// TIA Portal V17 export
// export: Created 2025-03-07T09:16:38.4737309Z, ExportSetting WithDefaults, DisplayName Totally Integrated Automation Portal, DisplayVersion V17 Update 8, DisplayName TIA Portal Openness, DisplayVersion V17 Update 8, DisplayName TIA Portal Version Control Interface, DisplayVersion V17, DisplayName SINAMICS Startdrive Advanced, DisplayVersion V17 SP2, DisplayName SINAMICS Startdrive G110M, G120, G120C, G120D, G120P, G115D, DisplayVersion V17 SP2, DisplayName SINAMICS Startdrive G130, G150, S120, S150, SINAMICS MV, S210, DisplayVersion V17 SP2, DisplayName STEP 7 Professional, DisplayVersion V17 Update 8, DisplayName SINUMERIK ONE STEP 7 Toolbox, DisplayVersion V17 Update 12, DisplayName SINUMERIK 840D sl STEP 7 Toolbox, DisplayVersion V17 Update 12, DisplayName STEP 7 Safety, DisplayVersion V17 Update 6, DisplayName WinCC Advanced, DisplayVersion V17 Update 8
DATA_BLOCK "DB2400_DBB_VALUES"   // DB2400
{ S7_Optimized_Access := 'FALSE'; DB_Accessible_From_OPC_UA := 'FALSE' }
AUTHOR : ETXETAR
VERSION : 1.0
// stored: AutoNumber false, DBAccessibleFromOPCUA false, DBAccessibleFromWebserver true, IsOnlyStoredInLoadMemory false, IsWriteProtectedInAS false
   VAR RETAIN
      DBB_DBW_DBD_VAL_0 : UInt := 0;   // MACHINE CNC CYCLE UNIT 01 STATION 0 ($A_DBB[0])
      DBB_DBW_DBD_VAL_1 : UInt := 1;
      DBB_DBW_DBD_VAL_2 : UInt := 2;   // MACHINE CNC CYCLE UNIT 01 STATION 3 ($A_DBB[2])
      DBB_DBW_DBD_VAL_3 : UInt := 3;
      DBB_DBW_DBD_VAL_4 : UInt := 4;   // MACHINE CNC CYCLE UNIT 01 STATION 4 ($A_DBB[4])
      DBB_DBW_DBD_VAL_5 : UInt := 5;
      DBB_DBW_DBD_VAL_6 : UInt := 6;   // MACHINE CNC CYCLE UNIT 02 STATION 0 ($A_DBB[6])
      DBB_DBW_DBD_VAL_7 : UInt := 7;
      DBB_DBW_DBD_VAL_8 : UInt := 8;   // MACHINE CNC CYCLE UNIT 02 STATION 2 ($A_DBB[8])
      DBB_DBW_DBD_VAL_9 : UInt := 9;
      DBB_DBW_DBD_VAL_10 : UInt := 10;   // MACHINE CNC CYCLE UNIT 02 STATION 3 ($A_DBB[9])
      DBB_DBW_DBD_VAL_11 : UInt := 11;
      DBB_DBW_DBD_VAL_12 : UInt := 12;   // MACHINE CNC CYCLE UNIT 02 STATION 4 ($A_DBB[9])
      DBB_DBW_DBD_VAL_14 : UInt := 14;   // MACHINE CNC CYCLE UNIT 03 STATION 0 ($A_DBB[14])
      DBB_DBW_DBD_VAL_19 : UInt := 19;
      DBB_DBW_DBD_VAL_20 : UInt := 20;   // FIXTURE NUMBER IN UNIT 01 STATION 1 ($A_DBB[20])
      DBB_DBW_DBD_VAL_22 : UInt := 22;   // FIXTURE NUMBER IN UNIT 02 STATION 1 ($A_DBB[22])
      DBB_DBW_DBD_VAL_23 : UInt := 23;
      DBB_DBW_DBD_VAL_24 : UInt := 24;
      DBB_DBW_DBD_VAL_30 : UInt := 30;   // PART TYPE ($A_DBB[30])
      DBB_DBW_DBD_VAL_31 : UInt := 31;
      DBB_DBW_DBD_VAL_34 : UInt := 34;
      DBB_DBW_DBD_VAL_35 : UInt := 35;
      DBB_DBW_DBD_VAL_40 : UInt := 40;   // FIXTURE 1 MACHINING MEMORY TO FULL DEPTH UNIT 01R ($A_DBB[40])
      DBB_DBW_DBD_VAL_41 : UInt := 41;   // FIXTURE 1 MACHINING MEMORY TO FULL DEPTH UNIT 01L ($A_DBB[41])
      DBB_DBW_DBD_VAL_44 : UInt := 44;   // FIXTURE 1 BACK CHAMFERS TRACER ($A_DBB[44])
      DBB_DBW_DBD_VAL_45 : UInt := 45;   // FIXTURE 1 TAPPING TRACER ($A_DBB[45])
      DBB_DBW_DBD_VAL_48 : UInt := 48;   // FIXTURE 2 MACHINING MEMORY TO FULL DEPTH UNIT 01R ($A_DBB[48])
      DBB_DBW_DBD_VAL_49 : UInt := 49;   // FIXTURE 2 MACHINING MEMORY TO FULL DEPTH UNIT 01L ($A_DBB[49])
      DBB_DBW_DBD_VAL_52 : UInt := 52;   // FIXTURE 2 BACK CHAMFERS TRACER ($A_DBB[52])
      DBB_DBW_DBD_VAL_53 : UInt := 53;   // FIXTURE 2 TAPPING TRACER ($A_DBB[53])
      DBB_DBW_DBD_VAL_56 : UInt := 56;   // FIXTURE 1 CLAMP STATUS ($A_DBB[56])
      DBB_DBW_DBD_VAL_57 : UInt := 57;   // FIXTURE 2 CLAMP STATUS ($A_DBB[57])
      DBB_DBW_DBD_VAL_58 : UInt := 58;   // PART SEATED CLAMP RECOVERY UNIT 01R ($A_DBB[58])
      DBB_DBW_DBD_VAL_59 : UInt := 59;   // PART SEATED CLAMP RECOVERY UNIT 01L ($A_DBB[59])
      DBB_DBW_DBD_VAL_60 : UInt := 60;   // AXIS W SAFETY MOVE ($A_DBB[60])
      DBB_DBW_DBD_VAL_61 : UInt := 61;   // AXIS B POSITIONS ($A_DBB[61])
      DBB_DBW_DBD_VAL_62 : UInt := 62;   // AXIS B IN POSITION TO LOAD ($A_DBB[62])
      DBB_DBW_DBD_VAL_64 : UInt := 64;   // MEASURE PROBE ALARM CODE ($A_DBB[64])
      DBB_DBW_DBD_VAL_65 : UInt := 65;   // MEASUREMENT FRECUENCY ($A_DBB[65])
      DBB_DBW_DBD_VAL_66 : UInt := 66;   // RESET GUD CYCLE VARIABLES ($A_DBB[66])
      DBB_DBW_DBD_VAL_67 : UInt := 67;   // CYCLE SELECTION CEMB ENABLE ($A_DBB[67])
      DBB_DBW_DBD_VAL_70 : UInt := 70;   // MQL VARIANT UNIT 01R ($A_DBB[70])
      DBB_DBW_DBD_VAL_71 : UInt := 71;   // MQL VARIANT UNIT 01L ($A_DBB[71])
      DBB_DBW_DBD_VAL_75 : UInt := 75;   // RFID ZONE TO WRITE IN TOOL HOLDER CHIP UNIT 01R ($A_DBB[75])
      DBB_DBW_DBD_VAL_76 : UInt := 76;   // RFID ZONE TO WRITE IN TOOL HOLDER CHIP UNIT 01L ($A_DBB[76])
      DBB_DBW_DBD_VAL_77 : UInt := 77;   // RFID ZONE TO WRITE IN TOOL HOLDER CHIP ($A_DBB[77])
      DBB_DBW_DBD_VAL_80 : UInt := 80;   // TAG ERROR UNIT 01R ($A_DBB[80])
      DBB_DBW_DBD_VAL_81 : UInt := 81;   // TAG ERROR UNIT 01L ($A_DBB[81])
      DBB_DBW_DBD_VAL_100 : UInt := 100;   // TOOL CLAMPING DIFFERENCE SP11 ($A_DBB[100])
      DBB_DBW_DBD_VAL_101 : UInt := 101;   // TOOL CLAMPING DIFFERENCE SP12 ($A_DBB[101])
      DBB_DBW_DBD_VAL_102 : UInt := 102;   // TOOL CLAMPING DIFFERENCE SP13 ($A_DBB[102])
      DBB_DBW_DBD_VAL_103 : UInt := 103;   // TOOL CLAMPING DIFFERENCE SP14 ($A_DBB[103])
      DBB_DBW_DBD_VAL_110 : UInt := 110;   // TOOL CLAMPING DIFFERENCE SP21 ($A_DBB[110])
      DBB_DBW_DBD_VAL_111 : UInt := 111;   // TOOL CLAMPING DIFFERENCE SP22 ($A_DBB[111])
      DBB_DBW_DBD_VAL_112 : UInt := 112;   // TOOL CLAMPING DIFFERENCE SP23 ($A_DBB[112])
      DBB_DBW_DBD_VAL_113 : UInt := 113;   // TOOL CLAMPING DIFFERENCE SP24 ($A_DBB[113])
      DBB_DBW_DBD_VAL_120 : UInt := 120;   // MAGAZINE MEMORY ALARM UNIT 01R ($A_DBB[120])
      DBB_DBW_DBD_VAL_121 : UInt := 121;   // MAGAZINE MEMORY ALARM TYPE UNIT 01R ($A_DBB[121])
      DBB_DBW_DBD_VAL_122 : UInt := 122;   // MAGAZINE TOOL FAULTED UNIT 01R ($A_DBB[122])
      DBB_DBW_DBD_VAL_123 : UInt := 123;   // MAGAZINE TOOL IN ERROR DATA UNIT 01R ($A_DBB[123])
      DBB_DBW_DBD_VAL_125 : UInt := 125;   // MAGAZINE MEMORY ALARM UNIT 01L ($A_DBB[125])
      DBB_DBW_DBD_VAL_126 : UInt := 126;   // MAGAZINE MEMORY ALARM TYPE UNIT 01L ($A_DBB[126])
      DBB_DBW_DBD_VAL_127 : UInt := 127;   // MAGAZINE TOOL FAULTED UNIT 01L ($A_DBB[127])
      DBB_DBW_DBD_VAL_128 : UInt := 128;   // MAGAZINE TOOL IN ERROR DATA UNIT 01L ($A_DBB[128])
      DBB_DBW_DBD_VAL_150 : UInt := 150;   // BK MIKRO MAGAZINE POSITION SP11 ($A_DBB[150])
      DBB_DBW_DBD_VAL_151 : UInt := 151;   // BK MIKRO MAGAZINE POSITION SP12 ($A_DBB[151])
      DBB_DBW_DBD_VAL_152 : UInt := 152;   // BK MIKRO MAGAZINE POSITION SP13 ($A_DBB[152])
      DBB_DBW_DBD_VAL_153 : UInt := 153;   // BK MIKRO MAGAZINE POSITION SP14 ($A_DBB[153])
      DBB_DBW_DBD_VAL_154 : UInt := 154;   // BK MIKRO MAGAZINE POSITION SP21 ($A_DBB[154])
      DBB_DBW_DBD_VAL_155 : UInt := 155;   // BK MIKRO MAGAZINE POSITION SP22 ($A_DBB[155])
      DBB_DBW_DBD_VAL_156 : UInt := 156;   // BK MIKRO MAGAZINE POSITION SP23 ($A_DBB[156])
      DBB_DBW_DBD_VAL_157 : UInt := 157;   // BK MIKRO MAGAZINE POSITION SP24 ($A_DBB[157])
      DBB_DBW_DBD_VAL_160 : UInt := 160;   // UNIT 01 POWDER FEEDER 1 CARRIER GAS NOMINAL LINE 1
      DBB_DBW_DBD_VAL_164 : UInt := 164;   // UNIT 01 POWDER FEEDER 1 CARRIER GAS NOMINAL LINE 2
      DBB_DBW_DBD_VAL_168 : UInt := 168;   // UNIT 01 POWDER FEEDER 1 DISK SPEED NOMINAL LINE 1
      DBB_DBW_DBD_VAL_172 : UInt := 172;   // UNIT 01 POWDER FEEDER 1 DISK SPEED NOMINAL LINE 2
      DBB_DBW_DBD_VAL_176 : UInt := 176;   // UNIT 01 POWDER FEEDER 1 STIRRER SPEED NOMINAL LINE 1
      DBB_DBW_DBD_VAL_180 : UInt := 180;   // UNIT 01 POWDER FEEDER 1 STIRRER SPEED NOMINAL LINE 2
      DBB_DBW_DBD_VAL_184 : UInt := 184;   // UNIT 01 POWDER FEEDER 1 HOPPER TEMPERATURE NOMINAL LINE 1
      DBB_DBW_DBD_VAL_188 : UInt := 188;   // UNIT 01 POWDER FEEDER 1 HOPPER TEMPERATURE NOMINAL LINE 2
      DBB_DBW_DBD_VAL_200 : UInt := 200;   // UNIT 02 POWDER FEEDER 1 CARRIER GAS NOMINAL LINE 1
      DBB_DBW_DBD_VAL_204 : UInt := 204;   // UNIT 02 POWDER FEEDER 1 CARRIER GAS NOMINAL LINE 2
      DBB_DBW_DBD_VAL_208 : UInt := 208;   // UNIT 02 POWDER FEEDER 1 DISK SPEED NOMINAL LINE 1
      DBB_DBW_DBD_VAL_212 : UInt := 212;   // UNIT 02 POWDER FEEDER 1 DISK SPEED NOMINAL LINE 2
      DBB_DBW_DBD_VAL_216 : UInt := 216;   // UNIT 02 POWDER FEEDER 1 STIRRER SPEED NOMINAL LINE 1
      DBB_DBW_DBD_VAL_220 : UInt := 220;   // UNIT 02 POWDER FEEDER 1 STIRRER SPEED NOMINAL LINE 2
      DBB_DBW_DBD_VAL_224 : UInt := 224;   // UNIT 02 POWDER FEEDER 1 HOPPER TEMPERATURE NOMINAL LINE 1
      DBB_DBW_DBD_VAL_228 : UInt := 228;   // UNIT 02 POWDER FEEDER 1 HOPPER TEMPERATURE NOMINAL LINE 2
      DBB_DBW_DBD_VAL_240 : UInt := 240;   // UNIT 02 POWDER FEEDER 2 CARRIER GAS NOMINAL LINE 1
      DBB_DBW_DBD_VAL_244 : UInt := 244;   // UNIT 02 POWDER FEEDER 2 CARRIER GAS NOMINAL LINE 2
      DBB_DBW_DBD_VAL_248 : UInt := 248;   // UNIT 02 POWDER FEEDER 2 DISK SPEED NOMINAL LINE 1
      DBB_DBW_DBD_VAL_252 : UInt := 252;   // UNIT 02 POWDER FEEDER 2 DISK SPEED NOMINAL LINE 2
      DBB_DBW_DBD_VAL_256 : UInt := 256;   // UNIT 02 POWDER FEEDER 2 STIRRER SPEED NOMINAL LINE 1
      DBB_DBW_DBD_VAL_260 : UInt := 260;   // UNIT 02 POWDER FEEDER 2 STIRRER SPEED NOMINAL LINE 2
      DBB_DBW_DBD_VAL_264 : UInt := 264;   // UNIT 02 POWDER FEEDER 2 HOPPER TEMPERATURE NOMINAL LINE 1
      DBB_DBW_DBD_VAL_268 : UInt := 268;   // UNIT 02 POWDER FEEDER 2 HOPPER TEMPERATURE NOMINAL LINE 2
      DBB_DBW_DBD_VAL_504 : UInt := 504;   // UNIT 01LASER POWER ($A_DBB[504])
      DBB_DBW_DBD_VAL_506 : UInt := 506;   // UNIT 01 LASER PROCESSING (0=CORE / 1=RING / 3=BRIGHTLINE WELD) ($A_DBB[506])
      DBB_DBW_DBD_VAL_508 : UInt := 508;   // UNIT 01 LASER POWER PORTION CORE (%) ($A_DBB[508])
      DBB_DBW_DBD_VAL_514 : UInt := 514;   // UNIT 02 LASER POWER ($A_DBB[514])
      DBB_DBW_DBD_VAL_516 : UInt := 516;   // UNIT 02 LASER PROCESSING (0=CORE / 1=RING / 3=BRIGHTLINE WELD) ($A_DBB[516])
      DBB_DBW_DBD_VAL_518 : UInt := 518;   // UNIT 02 LASER POWER PORTION CORE (%) ($A_DBB[518])
      DBB_DBW_DBD_VAL_1000 : UInt := 1000;   // UNIT 01 FIXTURE 1 PART A QUALITY STATUS ($A_DBB[1000])
      DBB_DBW_DBD_VAL_1001 : UInt := 1001;   // UNIT 01 FIXTURE 1 PART A PROCESS STATUS ($A_DBB[1001])
      DBB_DBW_DBD_VAL_1002 : UInt := 1002;   // UNIT 01 FIXTURE 1 PART C ($A_DBB[1002])
      DBB_DBW_DBD_VAL_1003 : UInt := 1003;   // UNIT 01 FIXTURE 1 PART D ($A_DBB[1003])
      DBB_DBW_DBD_VAL_1006 : UInt := 1006;   // UNIT 01 FIXTURE 2 PART A QUALITY STATUS ($A_DBB[1006])
      DBB_DBW_DBD_VAL_1007 : UInt := 1007;   // UNIT 01 FIXTURE 2 PART A PROCESS STATUS ($A_DBB[1007])
      DBB_DBW_DBD_VAL_1008 : UInt := 1008;   // UNIT 01 FIXTURE 2 PART C ($A_DBB[1008])
      DBB_DBW_DBD_VAL_1009 : UInt := 1009;   // UNIT 01 FIXTURE 2 PART D ($A_DBB[1009])
      DBB_DBW_DBD_VAL_1012 : UInt := 1012;   // UNIT 01 FIXTURE 3 PART A QUALITY STATUS ($A_DBB[1012])
      DBB_DBW_DBD_VAL_1013 : UInt := 1013;   // UNIT 01 FIXTURE 3 PART A PROCESS STATUS ($A_DBB[1013])
      DBB_DBW_DBD_VAL_1014 : UInt := 1014;   // UNIT 01 FIXTURE 3 PART C ($A_DBB[1014])
      DBB_DBW_DBD_VAL_1015 : UInt := 1015;   // UNIT 01 FIXTURE 3 PART D ($A_DBB[1015])
      DBB_DBW_DBD_VAL_1018 : UInt := 1018;   // UNIT 01 FIXTURE 4 PART A QUALITY STATUS ($A_DBB[1018])
      DBB_DBW_DBD_VAL_1019 : UInt := 1019;   // UNIT 01 FIXTURE 4 PART A PROCESS STATUS ($A_DBB[1019])
      DBB_DBW_DBD_VAL_1020 : UInt := 1020;   // UNIT 01 FIXTURE 4 PART C ($A_DBB[1020])
      DBB_DBW_DBD_VAL_1021 : UInt := 1021;   // UNIT 01 FIXTURE 4 PART D ($A_DBB[1021])
      DBB_DBW_DBD_VAL_1024 : UInt := 1024;   // UNIT 02 FIXTURE 1 PART A QUALITY STATUS ($A_DBB[1024])
      DBB_DBW_DBD_VAL_1025 : UInt := 1025;   // UNIT 02 FIXTURE 1 PART A PROCESS STATUS ($A_DBB[1025])
      DBB_DBW_DBD_VAL_1026 : UInt := 1026;   // UNIT 02 FIXTURE 1 PART C ($A_DBB[1026])
      DBB_DBW_DBD_VAL_1027 : UInt := 1027;   // UNIT 02 FIXTURE 1 PART D ($A_DBB[1027])
      DBB_DBW_DBD_VAL_1030 : UInt := 1030;   // UNIT 02 FIXTURE 2 PART A QUALITY STATUS ($A_DBB[1030])
      DBB_DBW_DBD_VAL_1031 : UInt := 1031;   // UNIT 02 FIXTURE 2 PART A PROCESS STATUS ($A_DBB[1031])
      DBB_DBW_DBD_VAL_1032 : UInt := 1032;   // UNIT 02 FIXTURE 2 PART C ($A_DBB[1032])
      DBB_DBW_DBD_VAL_1033 : UInt := 1033;   // UNIT 02 FIXTURE 2 PART D ($A_DBB[1033])
      DBB_DBW_DBD_VAL_1036 : UInt := 1036;   // UNIT 02 FIXTURE 3 PART A QUALITY STATUS ($A_DBB[1036])
      DBB_DBW_DBD_VAL_1037 : UInt := 1037;   // UNIT 02 FIXTURE 3 PART A PROCESS STATUS ($A_DBB[1037])
      DBB_DBW_DBD_VAL_1038 : UInt := 1038;   // UNIT 02 FIXTURE 3 PART C ($A_DBB[1038])
      DBB_DBW_DBD_VAL_1039 : UInt := 1039;   // UNIT 02 FIXTURE 3 PART D ($A_DBB[1039])
      DBB_DBW_DBD_VAL_1042 : UInt := 1042;   // UNIT 02 FIXTURE 4 PART A QUALITY STATUS ($A_DBB[1042])
      DBB_DBW_DBD_VAL_1043 : UInt := 1043;   // UNIT 02 FIXTURE 4 PART A PROCESS STATUS ($A_DBB[1043])
      DBB_DBW_DBD_VAL_1044 : UInt := 1044;   // UNIT 02 FIXTURE 4 PART C ($A_DBB[1044])
      DBB_DBW_DBD_VAL_1045 : UInt := 1045;   // UNIT 02 FIXTURE 4 PART D ($A_DBB[1045])
      DBB_DBW_DBD_VAL_1048 : UInt := 1048;   // UNIT 01 STATION 1 PART A QUALITY STATUS ($A_DBB[1048])
      DBB_DBW_DBD_VAL_1049 : UInt := 1049;   // UNIT 01 STATION 1 PART A PROCESS STATUS ($A_DBB[1049])
      DBB_DBW_DBD_VAL_1050 : UInt := 1050;   // UNIT 01 STATION 1 PART C ($A_DBB[1050])
      DBB_DBW_DBD_VAL_1051 : UInt := 1051;   // UNIT 01 STATION 1 PART D ($A_DBB[1051])
      DBB_DBW_DBD_VAL_1200 : UInt := 1200;   // CLEAN TOOL HOLDERS UNIT 01R ($A_DBB[1200])
      DBB_DBW_DBD_VAL_1201 : UInt := 1201;   // CLEAN TOOL HOLDERS SEQUENCE DONE UNIT 01R ($A_DBB[1201])
      DBB_DBW_DBD_VAL_1204 : UInt := 1204;   // CLEAN TOOL HOLDERS UNIT 01L ($A_DBB[1204])
      DBB_DBW_DBD_VAL_1205 : UInt := 1205;   // CLEAN TOOL HOLDERS SEQUENCE DONE UNIT 01L ($A_DBB[1205])
      DBB_DBW_DBD_VAL_1250 : UInt := 1250;   // WAIT CHANNEL 1 ($A_DBB[1250])
      DBB_DBW_DBD_VAL_1272 : UInt := 1272;   // UNIT 01 AXIS X13 ACTUAL SPEED ($A_DBB[1272])
      DBB_DBW_DBD_VAL_1276 : UInt := 1276;   // FIXTURE 1 PART A FLANGE Y ($A_DBB[1276])
      DBB_DBW_DBD_VAL_1280 : UInt := 1280;   // FIXTURE 1 PART A POST X ($A_DBB[1280])
      DBB_DBW_DBD_VAL_1284 : UInt := 1284;   // FIXTURE 1 PART A POST Y ($A_DBB[1284])
      DBB_DBW_DBD_VAL_1288 : UInt := 1288;   // FIXTURE 1 PART B FLANGE X ($A_DBB[1288])
      DBB_DBW_DBD_VAL_1292 : UInt := 1292;   // UNIT 01 SPINDLE C13 ACTUAL SPEED ($A_DBB[1292])
      DBB_DBW_DBD_VAL_1296 : UInt := 1296;   // FIXTURE 1 PART B POST X ($A_DBB[1296])
      DBB_DBW_DBD_VAL_1300 : UInt := 1300;   // FIXTURE 1 PART B POST Y ($A_DBB[1300])
      DBB_DBW_DBD_VAL_1352 : UInt := 1352;   // UNIT 02 AXIS X23 ACTUAL SPEED ($A_DBB[1352])
      DBB_DBW_DBD_VAL_1356 : UInt := 1356;   // FIXTURE 2 PART A FLANGE Y ($A_DBB[1356])
      DBB_DBW_DBD_VAL_1360 : UInt := 1360;   // FIXTURE 2 PART A POST X ($A_DBB[1360])
      DBB_DBW_DBD_VAL_1364 : UInt := 1364;   // FIXTURE 2 PART A POST Y ($A_DBB[1364])
      DBB_DBW_DBD_VAL_1368 : UInt := 1368;   // FIXTURE 2 PART B FLANGE X ($A_DBB[1368])
      DBB_DBW_DBD_VAL_1372 : UInt := 1372;   // UNIT 02 SPINDLE C23 ACTUAL SPEED ($A_DBB[1372])
      DBB_DBW_DBD_VAL_1376 : UInt := 1376;   // FIXTURE 2 PART B POST X ($A_DBB[1376])
      DBB_DBW_DBD_VAL_1380 : UInt := 1380;   // FIXTURE 2 PART B POST Y ($A_DBB[1380])
      DBB_DBW_DBD_VAL_1450 : UInt := 1450;   // NC TEST PROGRAM AXIS SELECTION ($A_DBB[1450])
      DBB_DBW_DBD_VAL_1452 : UInt := 1452;   // SERVICE POSITION PROGRAM SELECTION ($A_DBB[1452])
      DBB_DBW_DBD_VAL_1454 : UInt := 1454;   // SPEED FOR SP11. VIBRATION ANALYSIS ($A_DBB54
      DBB_DBW_DBD_VAL_1456 : UInt := 1456;   // SPEED FOR SP12. VIBRATION ANALYSIS ($A_DBB[1456])
      DBB_DBW_DBD_VAL_1458 : UInt := 1458;   // TIME FOR ANALYSIS. VIBRATION ANALYSIS UNIT 01R ($A_DBB[1458])
      DBB_DBW_DBD_VAL_1460 : UInt := 1460;   // TIME FOR START. VIBRATION ANALYSIS UNIT 01R ($A_DBB[1460])
      DBB_DBW_DBD_VAL_1462 : UInt := 1462;   // SPEED FOR SP21. VIBRATION ANALYSIS ($A_DBB[1462])
      DBB_DBW_DBD_VAL_1464 : UInt := 1464;   // SPEED FOR SP22. VIBRATION ANALYSIS ($A_DBB[1464])
      DBB_DBW_DBD_VAL_1466 : UInt := 1466;   // TIME FOR ANALYSIS. VIBRATION ANALYSIS UNIT 01L ($A_DBB[1466])
      DBB_DBW_DBD_VAL_1468 : UInt := 1468;   // TIME FOR START. VIBRATION ANALYSIS UNIT 01L ($A_DBB[1468])
      DBB_DBW_DBD_VAL_1500 : UInt := 1500;   // TOOL NAME. TOOL MAGAZINE 01R ($A_DBB[1500])
      DBB_DBW_DBD_VAL_1532 : UInt := 1532;   // DUPLO NUMBER. TOOL MAGAZINE 01R ($A_DBB[1532])
      DBB_DBW_DBD_VAL_1534 : UInt := 1534;   // LOCATION TYPE. TOOL MAGAZINE 01R ($A_DBB[1534])
      DBB_DBW_DBD_VAL_1536 : UInt := 1536;   // SIEMENS TOOL STATUS. TOOL MAGAZINE 01R ($A_DBB[1536])
      DBB_DBW_DBD_VAL_1538 : UInt := 1538;   // TYPE OF TOOL MONITORING. TOOL MAGAZINE 01R ($A_DBB[1538])
      DBB_DBW_DBD_VAL_1540 : UInt := 1540;   // CHECK TOOL BROKEN. TOOL MAGAZINE 01R ($A_DBB[1540])
      DBB_DBW_DBD_VAL_1542 : UInt := 1542;   // NUMBER OF CUTTING EDGES. TOOL MAGAZINE 01R ($A_DBB[1542])
      DBB_DBW_DBD_VAL_1544 : UInt := 1544;   // OEM 1. TOOL MAGAZINE 01R ($A_DBB[1544])
      DBB_DBW_DBD_VAL_1548 : UInt := 1548;   // OEM 2. TOOL MAGAZINE 01R ($A_DBB[1548])
      DBB_DBW_DBD_VAL_1552 : UInt := 1552;   // OEM 3. TOOL MAGAZINE 01R ($A_DBB[1552])
      DBB_DBW_DBD_VAL_1556 : UInt := 1556;   // OEM 4. TOOL MAGAZINE 01R ($A_DBB[1556])
      DBB_DBW_DBD_VAL_1560 : UInt := 1560;   // OEM 5. TOOL MAGAZINE 01R ($A_DBB[1560])
      DBB_DBW_DBD_VAL_1564 : UInt := 1564;   // OEM 6. TOOL MAGAZINE 01R ($A_DBB[1564])
      DBB_DBW_DBD_VAL_1568 : UInt := 1568;   // OEM 7. TOOL MAGAZINE 01R ($A_DBB[1568])
      DBB_DBW_DBD_VAL_1572 : UInt := 1572;   // OEM 8. TOOL MAGAZINE 01R ($A_DBB[1572])
      DBB_DBW_DBD_VAL_1576 : UInt := 1576;   // OEM 9. TOOL MAGAZINE 01R ($A_DBB[1576])
      DBB_DBW_DBD_VAL_1580 : UInt := 1580;   // OEM 10. TOOL MAGAZINE 01R ($A_DBB[1580])
      DBB_DBW_DBD_VAL_1584 : UInt := 1584;   // TOOL TYPE EDGE 1. TOOL MAGAZINE 01R ($A_DBB[1584])
      DBB_DBW_DBD_VAL_1586 : UInt := 1586;   // CUTTING POSITION EDGE 1. TOOL MAGAZINE 01R ($A_DBB[1586])
      DBB_DBW_DBD_VAL_1588 : UInt := 1588;   // TOOL LENGTH 1 EDGE 1. TOOL MAGAZINE 01R ($A_DBB[1588])
      DBB_DBW_DBD_VAL_1592 : UInt := 1592;   // TOOL LENGTH 2 EDGE 1. TOOL MAGAZINE 01R ($A_DBB[1592])
      DBB_DBW_DBD_VAL_1596 : UInt := 1596;   // TOOL LENGTH 3 EDGE 1. TOOL MAGAZINE 01R ($A_DBB[1596])
      DBB_DBW_DBD_VAL_1600 : UInt := 1600;   // TOOL RADIUS EDGE 1. TOOL MAGAZINE 01R ($A_DBB[1600])
      DBB_DBW_DBD_VAL_1604 : UInt := 1604;   // TOOL PITCH EDGE 1. TOOL MAGAZINE 01R ($A_DBB[1604])
      DBB_DBW_DBD_VAL_1608 : UInt := 1608;   // WEAR LENGTH EDGE 1. TOOL MAGAZINE 01R ($A_DBB[1608])
      DBB_DBW_DBD_VAL_1620 : UInt := 1620;   // WEAR RADIUS EDGE 1. TOOL MAGAZINE 01R ($A_DBB[1620])
      DBB_DBW_DBD_VAL_1645 : UInt := 1644;
      DBB_DBW_DBD_VAL_1644 : UInt := 1644;   // WARNING TOOL LIFE EDGE 1. TOOL MAGAZINE 01R ($A_DBB[1644])
      DBB_DBW_DBD_VAL_1648 : UInt := 1648;   // ACTUAL TOOL LIFE EDGE 1. TOOL MAGAZINE 01R ($A_DBB[1648])
      DBB_DBW_DBD_VAL_1652 : UInt := 1652;   // SET POINT QUANTITY EDGE 1. TOOL MAGAZINE 01R ($A_DBB[1652])
      DBB_DBW_DBD_VAL_1664 : UInt := 1664;   // TOOL TYPE EDGE 2. TOOL MAGAZINE 01R ($A_DBB[1664])
      DBB_DBW_DBD_VAL_1666 : UInt := 1666;   // CUTTING POSITION EDGE 2. TOOL MAGAZINE 01R ($A_DBB[1666])
      DBB_DBW_DBD_VAL_1668 : UInt := 1668;   // TOOL LENGTH 1 EDGE 2. TOOL MAGAZINE 01R ($A_DBB[1668])
      DBB_DBW_DBD_VAL_1672 : UInt := 1672;   // TOOL LENGTH 2 EDGE 2. TOOL MAGAZINE 01R ($A_DBB[1672])
      DBB_DBW_DBD_VAL_1676 : UInt := 1676;   // TOOL LENGTH 3 EDGE 2. TOOL MAGAZINE 01R ($A_DBB[1676])
      DBB_DBW_DBD_VAL_1680 : UInt := 1680;   // TOOL RADIUS EDGE 2. TOOL MAGAZINE 01R ($A_DBB[1680])
      DBB_DBW_DBD_VAL_1684 : UInt := 1684;   // TOOL PITCH EDGE 2. TOOL MAGAZINE 01R ($A_DBB[1684])
      DBB_DBW_DBD_VAL_1688 : UInt := 1688;   // WEAR LENGTH EDGE 2. TOOL MAGAZINE 01R ($A_DBB[1688])
      DBB_DBW_DBD_VAL_1700 : UInt := 1700;   // UNIT_01_NOOZLE_SURFACE_DISTANCE
      DBB_DBW_DBD_VAL_1704 : UInt := 1704;   // UNIT_02_NOOZLE_SURFACE_DISTANCE
      DBB_DBW_DBD_VAL_1724 : UInt := 1724;   // WARNING TOOL LIFE EDGE 2. TOOL MAGAZINE 01R ($A_DBB[1724])
      DBB_DBW_DBD_VAL_1728 : UInt := 1728;   // ACTUAL TOOL LIFE EDGE 2. TOOL MAGAZINE 01R ($A_DBB[1728])
      DBB_DBW_DBD_VAL_1732 : UInt := 1732;   // SET POINT QUANTITY EDGE 2. TOOL MAGAZINE 01R ($A_DBB[1732])
      DBB_DBW_DBD_VAL_1744 : UInt := 1744;   // TOOL TYPE EDGE 3. TOOL MAGAZINE 01R ($A_DBB[1744])
      DBB_DBW_DBD_VAL_1746 : UInt := 1746;   // CUTTING POSITION EDGE 3. TOOL MAGAZINE 01R ($A_DBB[1746])
      DBB_DBW_DBD_VAL_1748 : UInt := 1748;   // TOOL LENGTH 1 EDGE 3. TOOL MAGAZINE 01R ($A_DBB[1748])
      DBB_DBW_DBD_VAL_1752 : UInt := 1752;   // TOOL LENGTH 2 EDGE 3. TOOL MAGAZINE 01R ($A_DBB[1752])
      DBB_DBW_DBD_VAL_1756 : UInt := 1756;   // TOOL LENGTH 3 EDGE 3. TOOL MAGAZINE 01R ($A_DBB[1756])
      DBB_DBW_DBD_VAL_1760 : UInt := 1760;   // TOOL RADIUS EDGE 3. TOOL MAGAZINE 01R ($A_DBB[1760])
      DBB_DBW_DBD_VAL_1764 : UInt := 1764;   // TOOL PITCH EDGE 3. TOOL MAGAZINE 01R ($A_DBB[1764])
      DBB_DBW_DBD_VAL_1768 : UInt := 1768;   // WEAR LENGTH EDGE 3. TOOL MAGAZINE 01R ($A_DBB[1768])
      DBB_DBW_DBD_VAL_1780 : UInt := 1780;   // WEAR RADIUS EDGE 3. TOOL MAGAZINE 01R ($A_DBB[1780])
      DBB_DBW_DBD_VAL_1804 : UInt := 1804;   // WARNING TOOL LIFE EDGE 3. TOOL MAGAZINE 01R ($A_DBB[1804])
      DBB_DBW_DBD_VAL_1808 : UInt := 1808;   // ACTUAL TOOL LIFE EDGE 3. TOOL MAGAZINE 01R ($A_DBB[1808])
      DBB_DBW_DBD_VAL_1812 : UInt := 1812;   // SET POINT QUANTITY EDGE 3. TOOL MAGAZINE 01R ($A_DBB[1812])
      DBB_DBW_DBD_VAL_1824 : UInt := 1824;   // TOOL TYPE EDGE 4. TOOL MAGAZINE 01R ($A_DBB[1824])
      DBB_DBW_DBD_VAL_1826 : UInt := 1826;   // CUTTING POSITION EDGE 4. TOOL MAGAZINE 01R ($A_DBB[1826])
      DBB_DBW_DBD_VAL_1828 : UInt := 1828;   // TOOL LENGTH 1 EDGE 4. TOOL MAGAZINE 01R ($A_DBB[1828])
      DBB_DBW_DBD_VAL_1832 : UInt := 1832;   // TOOL LENGTH 2 EDGE 4. TOOL MAGAZINE 01R ($A_DBB[1832])
      DBB_DBW_DBD_VAL_1836 : UInt := 1836;   // TOOL LENGTH 3 EDGE 4. TOOL MAGAZINE ($A_DBB[1836])
      DBB_DBW_DBD_VAL_1840 : UInt := 1840;   // TOOL RADIUS EDGE 4. TOOL MAGAZINE 01R ($A_DBB[1840])
      DBB_DBW_DBD_VAL_1844 : UInt := 1844;   // TOOL PITCH EDGE 4. TOOL MAGAZINE 01R ($A_DBB[1844])
      DBB_DBW_DBD_VAL_1848 : UInt := 1848;   // WEAR LENGTH EDGE 4. TOOL MAGAZINE 01R ($A_DBB[1848])
      DBB_DBW_DBD_VAL_1860 : UInt := 1860;   // WEAR RADIUS EDGE 4. TOOL MAGAZINE 01R ($A_DBB[1860])
      DBB_DBW_DBD_VAL_1884 : UInt := 1884;   // WARNING TOOL LIFE EDGE 4. TOOL MAGAZINE 01R ($A_DBB[1884])
      DBB_DBW_DBD_VAL_1888 : UInt := 1888;   // ACTUAL TOOL LIFE EDGE 4. TOOL MAGAZINE 01R ($A_DBB[1888])
      DBB_DBW_DBD_VAL_1892 : UInt := 1892;   // SET POINT QUANTITY EDGE 4. TOOL MAGAZINE 01R ($A_DBB[1892])
      DBB_DBW_DBD_VAL_1904 : UInt := 1904;   // TOOL TYPE EDGE 5. TOOL MAGAZINE 01R ($A_DBB[1904])
      DBB_DBW_DBD_VAL_1906 : UInt := 1906;   // CUTTING POSITION EDGE 5. TOOL MAGAZINE 01R ($A_DBB[1906])
      DBB_DBW_DBD_VAL_1908 : UInt := 1908;   // TOOL LENGTH 1 EDGE 5. TOOL MAGAZINE 01R ($A_DBB[1908])
      DBB_DBW_DBD_VAL_1912 : UInt := 1912;   // TOOL LENGTH 2 EDGE 5. TOOL MAGAZINE 01R ($A_DBB[1912])
      DBB_DBW_DBD_VAL_1916 : UInt := 1916;   // TOOL LENGTH 3 EDGE 5. TOOL MAGAZINE 01R ($A_DBB[1916])
      DBB_DBW_DBD_VAL_1920 : UInt := 1920;   // TOOL RADIUS EDGE 5. TOOL MAGAZINE 01R ($A_DBB[1920])
      DBB_DBW_DBD_VAL_1924 : UInt := 1924;   // TOOL PITCH EDGE 5. TOOL MAGAZINE 01R ($A_DBB[1924])
      DBB_DBW_DBD_VAL_1928 : UInt := 1928;   // WEAR LENGTH EDGE 5. TOOL MAGAZINE 01R ($A_DBB[1928])
      DBB_DBW_DBD_VAL_1940 : UInt := 1940;   // WEAR RADIUS EDGE 5. TOOL MAGAZINE 01R ($A_DBB[1940])
      DBB_DBW_DBD_VAL_1964 : UInt := 1964;   // WARNING TOOL LIFE EDGE 5. TOOL MAGAZINE 01R ($A_DBB[1964])
      DBB_DBW_DBD_VAL_1968 : UInt := 1968;   // ACTUAL TOOL LIFE EDGE 5. TOOL MAGAZINE 01R ($A_DBB[1968])
      DBB_DBW_DBD_VAL_1972 : UInt := 1972;   // SET POINT QUANTITY EDGE 5. TOOL MAGAZINE 01R ($A_DBB[1972])
      DBB_DBW_DBD_VAL_1984 : UInt := 1984;   // GM SPINDLE NUMBER 01R ($A_DBB[1984])
      DBB_DBW_DBD_VAL_2000 : UInt := 2000;   // TOOL NAME. TOOL MAGAZINE 01L ($A_DBB[2000])
      DBB_DBW_DBD_VAL_2032 : UInt := 2032;   // DUPLO NUMBER. TOOL MAGAZINE 01L ($A_DBB[2032])
      DBB_DBW_DBD_VAL_2034 : UInt := 2034;   // LOCATION TYPE. TOOL MAGAZINE 01L ($A_DBB[2034])
      DBB_DBW_DBD_VAL_2036 : UInt := 2036;   // SIEMENS TOOL STATUS. TOOL MAGAZINE 01L ($A_DBB[2036])
      DBB_DBW_DBD_VAL_2038 : UInt := 2038;   // TYPE OF TOOL MONITORING. TOOL MAGAZINE 01L ($A_DBB[2038])
      DBB_DBW_DBD_VAL_2040 : UInt := 2040;   // CHECK TOOL BROKEN. TOOL MAGAZINE 01L ($A_DBB[2040])
      DBB_DBW_DBD_VAL_2042 : UInt := 2042;   // NUMBER OF CUTTING EDGES. TOOL MAGAZINE 01L ($A_DBB[2042])
      DBB_DBW_DBD_VAL_2044 : UInt := 2044;   // OEM 1. TOOL MAGAZINE 01L ($A_DBB[2044])
      DBB_DBW_DBD_VAL_2048 : UInt := 2048;   // OEM 2. TOOL MAGAZINE 01L ($A_DBB[2048])
      DBB_DBW_DBD_VAL_2052 : UInt := 2052;   // OEM 3. TOOL MAGAZINE 01L ($A_DBB[2052])
      DBB_DBW_DBD_VAL_2056 : UInt := 2056;   // OEM 4. TOOL MAGAZINE 01L ($A_DBB[2056])
      DBB_DBW_DBD_VAL_2060 : UInt := 2060;   // OEM 5. TOOL MAGAZINE 01L ($A_DBB[2060])
      DBB_DBW_DBD_VAL_2064 : UInt := 2064;   // OEM 6. TOOL MAGAZINE 01L ($A_DBB[2064])
      DBB_DBW_DBD_VAL_2068 : UInt := 2068;   // OEM 7. TOOL MAGAZINE 01L ($A_DBB[2068])
      DBB_DBW_DBD_VAL_2072 : UInt := 2072;   // OEM 8. TOOL MAGAZINE 01L ($A_DBB[2072])
      DBB_DBW_DBD_VAL_2076 : UInt := 2076;   // OEM 9. TOOL MAGAZINE 01L ($A_DBB[2076])
      DBB_DBW_DBD_VAL_2080 : UInt := 2080;   // OEM 10. TOOL MAGAZINE 01L ($A_DBB[2080])
      DBB_DBW_DBD_VAL_2084 : UInt := 2084;   // TOOL TYPE EDGE 1. TOOL MAGAZINE 01L ($A_DBB[2084])
      DBB_DBW_DBD_VAL_2086 : UInt := 2086;   // CUTTING POSITION EDGE 1. TOOL MAGAZINE 01L ($A_DBB[2086])
      DBB_DBW_DBD_VAL_2088 : UInt := 2088;   // TOOL LENGTH 1 EDGE 1. TOOL MAGAZINE 01L ($A_DBB[2088])
      DBB_DBW_DBD_VAL_2092 : UInt := 2092;   // TOOL LENGTH 2 EDGE 1. TOOL MAGAZINE 01L ($A_DBB[2092])
      DBB_DBW_DBD_VAL_2096 : UInt := 2096;   // TOOL LENGTH 3 EDGE 1. TOOL MAGAZINE 01L ($A_DBB[209])
      DBB_DBW_DBD_VAL_2100 : UInt := 2100;   // TOOL RADIUS EDGE 1. TOOL MAGAZINE 01L ($A_DBB[2100])
      DBB_DBW_DBD_VAL_2104 : UInt := 2104;   // TOOL PITCH EDGE 1. TOOL MAGAZINE 01L ($A_DBB[2104])
      DBB_DBW_DBD_VAL_2108 : UInt := 2108;   // WEAR LENGTH EDGE 1. TOOL MAGAZINE 01L ($A_DBB[2108])
      DBB_DBW_DBD_VAL_2120 : UInt := 2120;   // WEAR RADIUS EDGE 1. TOOL MAGAZINE 01L ($A_DBB[2120])
      DBB_DBW_DBD_VAL_2144 : UInt := 2144;   // WARNING TOOL LIFE EDGE 1. TOOL MAGAZINE 01L ($A_DBB[2144])
      DBB_DBW_DBD_VAL_2148 : UInt := 2148;   // ACTUAL TOOL LIFE EDGE 1. TOOL MAGAZINE 01L ($A_DBB[2148])
      DBB_DBW_DBD_VAL_2152 : UInt := 2152;   // SET POINT QUANTITY EDGE 1. TOOL MAGAZINE 01L ($A_DBB[2152])
      DBB_DBW_DBD_VAL_2164 : UInt := 2164;   // TOOL TYPE EDGE 2. TOOL MAGAZINE 01L ($A_DBB[2164])
      DBB_DBW_DBD_VAL_2166 : UInt := 2166;   // CUTTING POSITION EDGE 2. TOOL MAGAZINE 01L ($A_DBB[2166])
      DBB_DBW_DBD_VAL_2168 : UInt := 2168;   // TOOL LENGTH 1 EDGE 2. TOOL MAGAZINE 01L ($A_DBB[2168])
      DBB_DBW_DBD_VAL_2172 : UInt := 2172;   // TOOL LENGTH 2 EDGE 2. TOOL MAGAZINE 01L ($A_DBB[2172])
      DBB_DBW_DBD_VAL_2176 : UInt := 2176;   // TOOL LENGTH 3 EDGE 2. TOOL MAGAZINE 01L ($A_DBB[2176])
      DBB_DBW_DBD_VAL_2180 : UInt := 2180;   // TOOL RADIUS EDGE 2. TOOL MAGAZINE 01L ($A_DBB[2180])
      DBB_DBW_DBD_VAL_2184 : UInt := 2184;   // TOOL PITCH EDGE 2. TOOL MAGAZINE 01L ($A_DBB[2184])
      DBB_DBW_DBD_VAL_2188 : UInt := 2188;   // WEAR LENGTH EDGE 2. TOOL MAGAZINE 01L ($A_DBB[2188])
      DBB_DBW_DBD_VAL_2200 : UInt := 2200;   // WEAR RADIUS EDGE 2. TOOL MAGAZINE 01L ($A_DBB[2200])
      DBB_DBW_DBD_VAL_2224 : UInt := 2224;   // WARNING TOOL LIFE EDGE 2. TOOL MAGAZINE 01L ($A_DBB[2224])
      DBB_DBW_DBD_VAL_2228 : UInt := 2228;   // ACTUAL TOOL LIFE EDGE 2. TOOL MAGAZINE 01L ($A_DBB[2228])
      DBB_DBW_DBD_VAL_2232 : UInt := 2232;   // SET POINT QUANTITY EDGE 2. TOOL MAGAZINE 01L ($A_DBB[2232])
      DBB_DBW_DBD_VAL_2244 : UInt := 2244;   // TOOL TYPE EDGE 3. TOOL MAGAZINE 01L ($A_DBB[2244])
      DBB_DBW_DBD_VAL_2246 : UInt := 2246;   // CUTTING POSITION EDGE 3. TOOL MAGAZINE 01L ($A_DBB[2246])
      DBB_DBW_DBD_VAL_2248 : UInt := 2248;   // TOOL LENGTH 1 EDGE 3. TOOL MAGAZINE 01L ($A_DBB[2248])
      DBB_DBW_DBD_VAL_2252 : UInt := 2252;   // TOOL LENGTH 2 EDGE 3. TOOL MAGAZINE 01L ($A_DBB[2252])
      DBB_DBW_DBD_VAL_2256 : UInt := 2256;   // TOOL LENGTH 3 EDGE 3. TOOL MAGAZINE 01L ($A_DBB[2256])
      DBB_DBW_DBD_VAL_2260 : UInt := 2260;   // TOOL RADIUS EDGE 3. TOOL MAGAZINE 01L ($A_DBB[2260])
      DBB_DBW_DBD_VAL_2264 : UInt := 2264;   // TOOL PITCH EDGE 3. TOOL MAGAZINE 01L ($A_DBB[2264])
      DBB_DBW_DBD_VAL_2268 : UInt := 2268;   // WEAR LENGTH EDGE 3. TOOL MAGAZINE 01L ($A_DBB[2268])
      DBB_DBW_DBD_VAL_2280 : UInt := 2280;   // WEAR RADIUS EDGE 3. TOOL MAGAZINE 01L ($A_DBB[2280])
      DBB_DBW_DBD_VAL_2304 : UInt := 2304;   // WARNING TOOL LIFE EDGE 3. TOOL MAGAZINE 01L ($A_DBB[2304])
      DBB_DBW_DBD_VAL_2308 : UInt := 2308;   // ACTUAL TOOL LIFE EDGE 3. TOOL MAGAZINE 01L ($A_DBB[2308])
      DBB_DBW_DBD_VAL_2312 : UInt := 2312;   // SET POINT QUANTITY EDGE 3. TOOL MAGAZINE 01L ($A_DBB[2312])
      DBB_DBW_DBD_VAL_2324 : UInt := 2324;   // TOOL TYPE EDGE 4. TOOL MAGAZINE 01L ($A_DBB[2324])
      DBB_DBW_DBD_VAL_2326 : UInt := 2326;   // CUTTING POSITION EDGE 4. TOOL MAGAZINE 01L ($A_DBB[2326])
      DBB_DBW_DBD_VAL_2328 : UInt := 2328;   // TOOL LENGTH 1 EDGE 4. TOOL MAGAZINE 01L ($A_DBB[2328])
      DBB_DBW_DBD_VAL_2332 : UInt := 2332;   // TOOL LENGTH 2 EDGE 4. TOOL MAGAZINE 01L ($A_DBB[2332])
      DBB_DBW_DBD_VAL_2336 : UInt := 2336;   // TOOL LENGTH 3 EDGE 4. TOOL MAGAZINE 01L ($A_DBB[2336])
      DBB_DBW_DBD_VAL_2340 : UInt := 2340;   // TOOL RADIUS EDGE 4. TOOL MAGAZINE 01L ($A_DBB[2340])
      DBB_DBW_DBD_VAL_2344 : UInt := 2344;   // TOOL PITCH EDGE 4. TOOL MAGAZINE 01L ($A_DBB[2344])
      DBB_DBW_DBD_VAL_2348 : UInt := 2348;   // WEAR LENGTH EDGE 4. TOOL MAGAZINE 01L ($A_DBB[2348])
      DBB_DBW_DBD_VAL_2360 : UInt := 2360;   // WEAR RADIUS EDGE 4. TOOL MAGAZINE 01L ($A_DBB[2360])
      DBB_DBW_DBD_VAL_2384 : UInt := 2384;   // WARNING TOOL LIFE EDGE 4. TOOL MAGAZINE 01L ($A_DBB[2384])
      DBB_DBW_DBD_VAL_2388 : UInt := 2388;   // ACTUAL TOOL LIFE EDGE 4. TOOL MAGAZINE 01L ($A_DBB[2388])
      DBB_DBW_DBD_VAL_2392 : UInt := 2392;   // SET POINT QUANTITY EDGE 4. TOOL MAGAZINE 01L ($A_DBB[2392])
      DBB_DBW_DBD_VAL_2404 : UInt := 2404;   // TOOL TYPE EDGE 5. TOOL MAGAZINE 01L ($A_DBB[2404])
      DBB_DBW_DBD_VAL_2406 : UInt := 2406;   // CUTTING POSITION EDGE 5. TOOL MAGAZINE 01L ($A_DBB[2406])
      DBB_DBW_DBD_VAL_2408 : UInt := 2408;   // TOOL LENGTH 1 EDGE 5. TOOL MAGAZINE 01L ($A_DBB[2408])
      DBB_DBW_DBD_VAL_2412 : UInt := 2412;   // TOOL LENGTH 2 EDGE 5. TOOL MAGAZINE 01L ($A_DBB[2412])
      DBB_DBW_DBD_VAL_2416 : UInt := 2416;   // TOOL LENGTH 3 EDGE 5. TOOL MAGAZINE 01L ($A_DBB[2416])
      DBB_DBW_DBD_VAL_2420 : UInt := 2420;   // TOOL RADIUS EDGE 5. TOOL MAGAZINE 01L ($A_DBB[2420])
      DBB_DBW_DBD_VAL_2424 : UInt := 2424;   // TOOL PITCH EDGE 5. TOOL MAGAZINE 01L ($A_DBB[2424)
      DBB_DBW_DBD_VAL_2428 : UInt := 2428;   // WEAR LENGTH EDGE 5. TOOL MAGAZINE 01L ($A_DBB[2428])
      DBB_DBW_DBD_VAL_2440 : UInt := 2440;   // WEAR RADIUS EDGE 5. TOOL MAGAZINE 01L ($A_DBB[2440])
      DBB_DBW_DBD_VAL_2464 : UInt := 2464;   // WARNING TOOL LIFE EDGE 5. TOOL MAGAZINE 01L ($A_DBB[2464])
      DBB_DBW_DBD_VAL_2468 : UInt := 2468;   // ACTUAL TOOL LIFE EDGE 5. TOOL MAGAZINE 01L ($A_DBB[2468])
      DBB_DBW_DBD_VAL_2472 : UInt := 2472;   // SET POINT QUANTITY EDGE 5. TOOL MAGAZINE 01L ($A_DBB[2472])
      DBB_DBW_DBD_VAL_2484 : UInt := 2484;   // GM SPINDLE NUMBER 01L ($A_DBB[2484])
      DBB_DBW_DBD_VAL_3000 : UInt := 3000;   // CRASH BORE MEASURE POINT 1 ($A_DBB[3000])
      DBB_DBW_DBD_VAL_3004 : UInt := 3004;   // CRASH BORE MEASURE POINT 2 ($A_DBB[3004])
      DBB_DBW_DBD_VAL_3008 : UInt := 3008;   // CRASH BORE MEASURE POINT 3 ($A_DBB[3008])
      DBB_DBW_DBD_VAL_3012 : UInt := 3012;   // CRASH BORE MEASURE POINT 4 ($A_DBB3012)]
      DBB_DBW_DBD_VAL_3016 : UInt := 3016;   // CRASH BORE MEASURE POINT 5 ($A_DBB[3016])
      DBB_DBW_DBD_VAL_3020 : UInt := 3020;   // CRASH BORE MEASURE POINT 6 ($A_DBB[3020])
      DBB_DBW_DBD_VAL_3024 : UInt := 3024;   // CRASH BORE MEASURE POINT 7X ($A_DBB[3024])
      DBB_DBW_DBD_VAL_3028 : UInt := 3028;   // CRASH BORE MEASURE POINT 7Y ($A_DBB[3028])
      DBB_DBW_DBD_VAL_3032 : UInt := 3032;   // CRASH BORE MEASURE POINT 8X ($A_DBB[3032])
      DBB_DBW_DBD_VAL_3036 : UInt := 3036;   // CRASH BORE MEASURE POINT 8Y ($A_DBB[3036])
      DBB_DBW_DBD_VAL_3200 : UInt := 3200;   // MEASURING PROBE PART A 1 ($A_DBB[3200])
      DBB_DBW_DBD_VAL_3204 : UInt := 3204;   // MEASURING PROBE PART A 2 ($A_DBB[3204])
      DBB_DBW_DBD_VAL_3208 : UInt := 3208;   // MEASURING PROBE PART B 1 ($A_DBB[3208])
      DBB_DBW_DBD_VAL_3212 : UInt := 3212;   // MEASURING PROBE PART B 2 ($A_DBB[3212])
      DBB_DBW_DBD_VAL_3216 : UInt := 3216;   // MEASURING PROBE PART C 1 ($A_DBB[3216])
      DBB_DBW_DBD_VAL_3220 : UInt := 3220;   // MEASURING PROBE PART C 2 ($A_DBB[3220])
      DBB_DBW_DBD_VAL_3224 : UInt := 3224;   // MEASURING PROBE PART A1 1 ($A_DBB[3224])
      DBB_DBW_DBD_VAL_3228 : UInt := 3228;   // MEASURING PROBE PART A1 2 ($A_DBB[3228])
      DBB_DBW_DBD_VAL_3232 : UInt := 3232;   // MEASURING PROBE PART B1 1 ($A_DBB[3232])
      DBB_DBW_DBD_VAL_3236 : UInt := 3236;   // MEASURING PROBE PART B1 2 ($A_DBB[3236])
      DBB_DBW_DBD_VAL_3240 : UInt := 3240;   // MEASURING PROBE PART C1 1 ($A_DBB[3240])
      DBB_DBW_DBD_VAL_3244 : UInt := 3244;   // MEASURING PROBE PART C1 2 ($A_DBB[3244])
      DBB_DBW_DBD_VAL_3248 : UInt := 3248;   // MEASURING PROBE PART A2 1 ($A_DBB[3248])
      DBB_DBW_DBD_VAL_3252 : UInt := 3252;   // MEASURING PROBE PART A2 2 ($A_DBB[3252])
      DBB_DBW_DBD_VAL_3256 : UInt := 3256;   // MEASURING PROBE PART B2 1 ($A_DBB[3256])
      DBB_DBW_DBD_VAL_3260 : UInt := 3260;   // MEASURING PROBE PART B2 2 ($A_DBB[3260])
      DBB_DBW_DBD_VAL_3264 : UInt := 3264;   // MEASURING PROBE PART C2 1 ($A_DBB[3264])
      DBB_DBW_DBD_VAL_3268 : UInt := 3268;   // MEASURING PROBE PART C2 2 ($A_DBB[3268])
      DBB_DBW_DBD_VAL_3400 : UInt := 3400;   // TORQUE AXIS SP11 ($A_DBB[3400])
      DBB_DBW_DBD_VAL_3404 : UInt := 3404;   // TORQUE AXIS SP12 ($A_DBB[3404])
      DBB_DBW_DBD_VAL_3408 : UInt := 3408;   // TORQUE AXIS SP13 ($A_DBB[3408])
      DBB_DBW_DBD_VAL_3412 : UInt := 3412;   // TORQUE AXIS SP14 ($A_DBB[3412])
      DBB_DBW_DBD_VAL_3416 : UInt := 3416;   // TORQUE AXIS SP15 ($A_DBB[3416])
      DBB_DBW_DBD_VAL_3420 : UInt := 3420;   // TORQUE AXIS SP16 ($A_DBB[3420])
      DBB_DBW_DBD_VAL_3424 : UInt := 3424;   // TORQUE AXIS SP21 ($A_DBB[3424])
      DBB_DBW_DBD_VAL_3428 : UInt := 3428;   // TORQUE AXIS SP22 ($A_DBB[3428])
      DBB_DBW_DBD_VAL_3432 : UInt := 3432;   // TORQUE AXIS SP23 ($A_DBB[3432])
      DBB_DBW_DBD_VAL_3436 : UInt := 3436;   // TORQUE AXIS SP24 ($A_DBB[3436])
      DBB_DBW_DBD_VAL_3440 : UInt := 3440;   // TORQUE AXIS SP25 ($A_DBB[3440])
      DBB_DBW_DBD_VAL_3444 : UInt := 3444;   // TORQUE AXIS SP26 ($A_DBB[3444])
      DBB_DBW_DBD_VAL_3448 : UInt := 3448;   // TORQUE AXIS Z11 ($A_DBB[3448])
      DBB_DBW_DBD_VAL_3452 : UInt := 3452;   // TORQUE AXIS Z12 ($A_DBB[3452])
      DBB_DBW_DBD_VAL_3456 : UInt := 3456;   // TORQUE AXIS Z13 ($A_DBB[3456])
      DBB_DBW_DBD_VAL_3460 : UInt := 3460;   // TORQUE AXIS Z14 ($A_DBB[3460])
      DBB_DBW_DBD_VAL_3464 : UInt := 3464;   // TORQUE AXIS Z21 ($A_DBB[3464])
      DBB_DBW_DBD_VAL_3468 : UInt := 3468;   // TORQUE AXIS Z22 ($A_DBB[3468])
      DBB_DBW_DBD_VAL_3472 : UInt := 3472;   // TORQUE AXIS Z23 ($A_DBB[3472])
      DBB_DBW_DBD_VAL_3476 : UInt := 3476;   // TORQUE AXIS Z24 ($A_DBB[3476])
   END_VAR
BEGIN
END_DATA_BLOCK
